// TIA Portal V16 export
// export: Created 2021-09-08T12:46:15.6423288Z, ExportSetting WithDefaults, DisplayName Totally Integrated Automation Portal, DisplayVersion V16 Update 3, DisplayName TIA Portal Version Control Interface, DisplayVersion V16 Update 2, DisplayName TIA Portal Openness, DisplayVersion V16 Update 3, DisplayName TIA Portal Teamcenter Gateway, DisplayVersion V16, DisplayName STEP 7 Professional, DisplayVersion V16 Update 3, DisplayName STEP 7 Safety, DisplayVersion V16, DisplayName WinCC Advanced, DisplayVersion V16 Update 3
DATA_BLOCK "hardwareTimePulse_DB"   // DB13
VERSION : 0.1
// stored: AutoNumber true, DBAccessibleFromOPCUA true, InstanceOfName hardwareTimePulse, InstanceOfType FB
"hardwareTimePulse"
   // VAR
   //    pTrig1HZ : Bool;
   //    pTrig05Hz : Bool;
   //    pTrig0625Hz : Bool;
   //    pTrig1_25HZ : Bool;
   //    pTrig2HZ : Bool;
   //    pTrig2_5Hz : Bool;
   //    pTirg5Hz : Bool;
   //    pTrig10Hz : Bool;
   // END_VAR
BEGIN
END_DATA_BLOCK
